// TwinCAT 3 PLC project Untitled1
// ProgramVersion: 3.1.4026.17
// libraries:
//   Tc2_Standard, * (Beckhoff Automation GmbH)
//   Tc2_System, * (Beckhoff Automation GmbH)
// project tree:
//   DUTs/ Box_Phase.TcDUT, Lay_Phase.TcDUT, Pal_Phase.TcDUT
//   GVLs/ GVL.TcGVL
//   / PlcTask.TcTTO
//   POUs/ BoxAccum.TcPOU, LayerPlace.TcPOU, MAIN.TcPOU, Pallet.TcPOU
// real-time tasks:
//   TASK PlcTask: cycle T#10ms, priority 20, ADS port 350

CONFIGURATION Untitled1
    RESOURCE PLC ON TwinCAT3
        TASK PlcTask(INTERVAL := T#10ms, PRIORITY := 20);
        PROGRAM MAIN WITH PlcTask : MAIN;
    END_RESOURCE
END_CONFIGURATION

// ---- DUTs/Box_Phase.TcDUT
{attribute 'qualified_only'}
{attribute 'strict'}
{attribute 'to_string'}
TYPE Box_Phase :
(
	Start, Run, Delay, PushFall, PushRise, TargetCheck, Clamp, Drop, Hold 
);
END_TYPE

// ---- DUTs/Lay_Phase.TcDUT
{attribute 'qualified_only'}
{attribute 'strict'}
{attribute 'to_string'}
TYPE Lay_Phase :
(
	Start,Down, LayCheck, ElvLim, ElvNex, ElvDone
):=Start;
END_TYPE

// ---- DUTs/Pal_Phase.TcDUT
{attribute 'qualified_only'}
{attribute 'strict'}
{attribute 'to_string'}
TYPE Pal_Phase :
(
	idle, Loaded, Ready_for_Boxes, Box_Loaded, Ready_for_Disp, Paused
) :=idle;
END_TYPE

// ---- GVLs/GVL.TcGVL
{attribute 'qualified_only'}
VAR_GLOBAL
    // Runtime State
    ePal_Phase              : Pal_Phase;  // Pallet machine phase
    bRunning                : BOOL;       // Line is running
    bFinishing              : BOOL;       // Graceful stop in progress
    bLayCheck               : BOOL;

    // Actuator Requests (to be AND-masked with bEnable before FIO outputs)
    // Conveyors & Belts 
    req_M010_CONV_Entry        : BOOL;
    req_M020_CONV_Incl         : BOOL;
    req_M031_CONV_PalBelt_FWD  : BOOL;
    req_M032_CONV_PalBelt_BCK  : BOOL;
    req_M080_CONV_Roll         : BOOL;
    req_M100_CONV_Exit         : BOOL;

    // Pusher / Turn / Clamp / Plate 
    req_M040_ARM_PalPush       : BOOL;
    req_M041_ARM_PalTurn       : BOOL;
    req_M050_CLAMP_Pal         : BOOL;	
    req_M050_CLAMP_Pal_B       : BOOL;
    req_M050_CLAMP_Pal_L       : BOOL;	
    req_M060_PLATE_Pal         : BOOL;     
    req_M060_PLATE_Pal_B       : BOOL;
    req_M060_PLATE_Pal_L       : BOOL;	

    // Elevator 
    req_M071_ELEV_Pal_UP       : BOOL;
    req_M072_ELEV_Pal_DOWN     : BOOL;
    req_M073_ELEV_Pal_M2LIM    : BOOL;  	
    req_M073_ELEV2TOP          : BOOL;   // move elevator to TOP 
    req_M073_ELEV2Bottom       : BOOL;   // move elevator to BOTTOM 

    // Pallet Chain
    req_M091_CONV_PalChain_FWD : BOOL;

    // Light
    req_P060_Light_SPPlus      : BOOL;   // Stack light: SP+
    req_P070_Light_SPMinus     : BOOL;   // Stack light: SP-
END_VAR

// ---- POUs/MAIN.TcPOU
PROGRAM MAIN
VAR
    // ACTUATORS (Outputs to field)
    FIO_M010_CONV_Entry          : BOOL;
    FIO_M020_CONV_Incl           : BOOL;
    FIO_M031_CONV_PalBelt_FWD    : BOOL;
    FIO_M032_CONV_PalBelt_BCK    : BOOL;
    FIO_M040_ARM_PalPush         : BOOL;
    FIO_M050_CLAMP_Pal           : BOOL;
    FIO_M060_PLATE_Pal           : BOOL;
    FIO_M071_ELEV_Pal_UP         : BOOL;
    FIO_M072_ELEV_Pal_DOWN       : BOOL;
    FIO_M073_ELEV_Pal_M2LIM      : BOOL;
    FIO_M080_CONV_Roll           : BOOL;
    FIO_M091_CONV_PalChain_FWD   : BOOL;
    FIO_M100_CONV_Exit           : BOOL;

    // SENSORS (Inputs from field)
    FIO_B010_PallClamped         : BOOL;        // Clamp sensor
    FIO_B020_PallPlateLim        : BOOL := TRUE; // NC: Plate limit (healthy=TRUE)
    FIO_B030_PallPushLim         : BOOL := TRUE; // NC: Pusher home limit (healthy=TRUE)
    FIO_B040_PallElvMov          : BOOL;        // Elevator motion status
    FIO_B050_PallElvFrLim        : BOOL;        // Elevator front/top limit
    FIO_B060_PallElvBckLim       : BOOL;        // Elevator back/bottom limit
    FIO_B070_PallReflexCnt       : BOOL := TRUE; // NC: Box counter reflex (healthy=TRUE)

    // BUTTONS 
    FIO_S100_EStop               : BOOL := TRUE; // NC: Emergency stop (healthy=TRUE)
    FIO_S010_Start               : BOOL;         // Start push button
    FIO_S020_Stop                : BOOL := TRUE; // NC: Stop push button (healthy=TRUE)
    FIO_S040_IN_LaySP_PLUS       : BOOL;         // HMI: Layer SP +
    FIO_S050_IN_LaySP_MINUS      : BOOL;         // HMI: Layer SP -

    // DISPLAYS / PROCESS VALUES (to HMI)
    // Consider RETAIN/PERSISTENT for setpoints if needed across reboots.
    FIO_P010_iPallID             : INT  := 0;   // Pallet ID
    FIO_P020_iLayCur             : INT  := 1;   // Current layer (1..10)
    FIO_P030_iLaySP              : INT  := 1;   // Layer setpoint (1..10)
    FIO_P040_Light_Start         : BOOL;        // Stack light: Start
    FIO_P050_Light_Stop          : BOOL;        // Stack light: Stop
    FIO_P060_Light_SPPlus        : BOOL;        // Stack light: SP+
    FIO_P070_Light_SPMinus       : BOOL;        // Stack light: SP-

    // FUNCTION BLOCK INSTANCES
    fbPallet		             : Pallet;
    fbBoxAccum                   : BoxAccum;
    fbLayerPlace                 : LayerPlace;


	// EDGE DETECTORS / LATCHES / FLAGS
    rStart                       : R_TRIG;      // Rising-edge detector for Start
    fStop                        : F_TRIG;      // Falling-edge detector for Stop
    fRunFall                     : F_TRIG;      // Falling-edge detector for bRunning
    srRunning                    : SR;          // Set/Reset latch for running state
    bEstopActive                 : BOOL;        // TRUE when Estop is active
END_VAR

// Structure: Safety → FBs → State → Requests → Actuators + Light

// SAFETY & RUN CONTROL
// Emergency stop
bEstopActive := NOT FIO_S100_EStop;     // TRUE = Estop pressed

// Start / Stop edge detection
rStart(CLK := FIO_S010_Start);
fStop (CLK := FIO_S020_Stop);

// SR latch for Running status
srRunning(
    SET1  := rStart.Q AND NOT bEstopActive,
    RESET := fStop.Q
);

// Running / Finishing flags 
IF srRunning.Q1 THEN
    gvl.bRunning   := TRUE;             // Enter RUN
    gvl.bFinishing := FALSE;            // Reset finishing
ELSE
    gvl.bRunning := FALSE;
END_IF

// Detect normal stop (falling edge of Running) 
fRunFall(CLK := gvl.bRunning);
IF (NOT bEstopActive) AND fRunFall.Q THEN
    gvl.bFinishing := TRUE;             // Controlled stop sequence
END_IF

//Estop clears finishing immediately
IF bEstopActive THEN
    gvl.bFinishing := FALSE;
END_IF

// FUNCTION BLOCK CALLS

fbPallet(
    PallElvFrLim := FIO_B050_PallElvFrLim,
    PallElvBckLim:= FIO_B060_PallElvBckLim,
    PallElvMov   := FIO_B040_PallElvMov,
    iPallID      => FIO_P010_iPallID
);

fbBoxAccum(
    PallClamped      := FIO_B010_PallClamped,
    PallPlateLim_NC  := FIO_B020_PallPlateLim,
    PallPushLim      := FIO_B030_PallPushLim,
    PallReflexCnt_NC := FIO_B070_PallReflexCnt
);

fbLayerPlace(
    LaySP_PLUS       := FIO_S040_IN_LaySP_PLUS,
    LaySP_MINUS      := FIO_S050_IN_LaySP_MINUS,
    PallElvMov       := FIO_B040_PallElvMov,
    iLaySP           => FIO_P030_iLaySP,
    iLayCur          => FIO_P020_iLayCur
);

// STATE → REQUESTS
// Translate pallet phase into actuator requests
CASE gvl.ePal_Phase OF

    Pal_Phase.Loaded:
        gvl.req_M073_ELEV_Pal_M2LIM := gvl.req_M073_ELEV2TOP;

    Pal_Phase.Ready_for_Boxes:
        gvl.req_M073_ELEV_Pal_M2LIM := gvl.req_M073_ELEV2Bottom;
        gvl.req_M050_CLAMP_Pal      := gvl.req_M050_CLAMP_Pal_B;
        gvl.req_M060_PLATE_Pal      := gvl.req_M050_CLAMP_Pal_B;

    Pal_Phase.Box_Loaded:
        gvl.req_M050_CLAMP_Pal      := gvl.req_M050_CLAMP_Pal_L;
        gvl.req_M060_PLATE_Pal      := gvl.req_M050_CLAMP_Pal_L;

ELSE
    gvl.req_M073_ELEV_Pal_M2LIM    := FALSE;
    gvl.req_M050_CLAMP_Pal         := FALSE;
    gvl.req_M060_PLATE_Pal         := FALSE;
END_CASE;

// REQUESTS → ACTUATORS
// Reset all outputs (avoid stale signals)
FIO_M010_CONV_Entry        := FALSE;
FIO_M020_CONV_Incl         := FALSE;
FIO_M031_CONV_PalBelt_FWD  := FALSE;
FIO_M032_CONV_PalBelt_BCK  := FALSE;
FIO_M040_ARM_PalPush       := FALSE;
FIO_M050_CLAMP_Pal         := FALSE;
FIO_M060_PLATE_Pal         := FALSE;
FIO_M071_ELEV_Pal_UP       := FALSE;
FIO_M072_ELEV_Pal_DOWN     := FALSE;
FIO_M073_ELEV_Pal_M2LIM    := FALSE;
FIO_M080_CONV_Roll         := FALSE;
FIO_M091_CONV_PalChain_FWD := FALSE;
FIO_M100_CONV_Exit         := FALSE;

// Map all requests to outputs (with Estop interlock)
FIO_M010_CONV_Entry        := gvl.req_M010_CONV_Entry        AND NOT bEstopActive;
FIO_M020_CONV_Incl         := gvl.req_M020_CONV_Incl         AND NOT bEstopActive;
FIO_M031_CONV_PalBelt_FWD  := gvl.req_M031_CONV_PalBelt_FWD  AND NOT bEstopActive;
FIO_M032_CONV_PalBelt_BCK  := gvl.req_M032_CONV_PalBelt_BCK  AND NOT bEstopActive;
FIO_M040_ARM_PalPush       := gvl.req_M040_ARM_PalPush       AND NOT bEstopActive;
FIO_M050_CLAMP_Pal         := gvl.req_M050_CLAMP_Pal         AND NOT bEstopActive;
FIO_M060_PLATE_Pal         := gvl.req_M060_PLATE_Pal         AND NOT bEstopActive;
FIO_M071_ELEV_Pal_UP       := gvl.req_M071_ELEV_Pal_UP       AND NOT bEstopActive;
FIO_M072_ELEV_Pal_DOWN     := gvl.req_M072_ELEV_Pal_DOWN     AND NOT bEstopActive;
FIO_M080_CONV_Roll         := gvl.req_M080_CONV_Roll         AND NOT bEstopActive;
FIO_M091_CONV_PalChain_FWD := gvl.req_M091_CONV_PalChain_FWD AND NOT bEstopActive;
FIO_M100_CONV_Exit         := gvl.req_M100_CONV_Exit         AND NOT bEstopActive;
FIO_M073_ELEV_Pal_M2LIM    := gvl.req_M073_ELEV_Pal_M2LIM    AND NOT bEstopActive;

// Light
FIO_P040_Light_Start       := srRunning.Q1;
FIO_P050_Light_Stop        := gvl.bFinishing;
FIO_P060_Light_SPPlus      := gvl.req_P060_Light_SPPlus;
FIO_P070_Light_SPMinus     := gvl.req_P070_Light_SPMinus;

END_PROGRAM

// ---- POUs/Pallet.TcPOU
FUNCTION_BLOCK Pallet
VAR_INPUT
    // Sensors 
    PallElvFrLim   : BOOL;   // Front limit switch
    PallElvBckLim  : BOOL;   // Back limit switch
    PallElvMov     : BOOL;   // Elevator in motion (TRUE while moving)
END_VAR

VAR_OUTPUT
    iPallID        : INT := 0;
END_VAR

VAR
    // Edge detectors
    rPallElvBckLim : R_TRIG;
    rPallElvFrLim  : R_TRIG;
    fPallElvMov    : F_TRIG;
    fPallElvFrLim  : F_TRIG;

    // Latches (SR)
    srCONV_Roll         : SR;
    srCONV_PalChain_FWD : SR;
    srELEV_Pal_UP       : SR;
END_VAR

// Edge detection 
rPallElvBckLim (CLK := PallElvBckLim);   // rising: pallet tail hits back limit
rPallElvFrLim  (CLK := PallElvFrLim);    // rising: pallet head hits front limit
fPallElvMov    (CLK := PallElvMov);      // falling: elevator motion stopped
fPallElvFrLim  (CLK := PallElvFrLim);    // falling: pallet clears front

// Safe defaults each scan
gvl.req_M080_CONV_Roll         := FALSE;
gvl.req_M091_CONV_PalChain_FWD := FALSE;    
gvl.req_M071_ELEV_Pal_UP       := FALSE;
gvl.req_M073_ELEV2TOP          := FALSE;
gvl.req_M073_ELEV_Pal_M2LIM    := FALSE;
gvl.req_M100_CONV_Exit         := FALSE;

CASE gvl.ePal_Phase OF

    // idle → load pallet
    Pal_Phase.idle:

        // Roller runs while no limits; stop on front-limit rising or stop command
        srCONV_Roll(
            SET1  := gvl.bRunning AND (NOT PallElvFrLim) AND (NOT PallElvBckLim),
            RESET := rPallElvFrLim.Q
        );
        gvl.req_M080_CONV_Roll := srCONV_Roll.Q1;
        gvl.req_M100_CONV_Exit := srCONV_Roll.Q1;

        // Chain IN: start when back-limit is hit; stop on front-limit rising or stop
        srCONV_PalChain_FWD(
            SET1  := rPallElvBckLim.Q,
            RESET := rPallElvFrLim.Q
        );
        gvl.req_M091_CONV_PalChain_FWD := srCONV_PalChain_FWD.Q1;

        // Pallet ID
        IF rPallElvBckLim.Q THEN 
            iPallID := iPallID + 10;
        END_IF

        // Transition to Loaded when both limits are TRUE
        IF PallElvFrLim AND PallElvBckLim THEN
            gvl.ePal_Phase := Pal_Phase.Loaded;
        END_IF

    // Loaded → move elevator up to the top
    Pal_Phase.Loaded:

        // Latch UP; reset when motion stops (reached top) or stop command
        srELEV_Pal_UP(
            SET1  := TRUE,       
            RESET := fPallElvMov.Q
        );
        gvl.req_M071_ELEV_Pal_UP := srELEV_Pal_UP.Q1;
        gvl.req_M073_ELEV2TOP    := srELEV_Pal_UP.Q1;   // same intent signal

        // When motion stops, elevator is at top
        IF fPallElvMov.Q THEN
            gvl.ePal_Phase := Pal_Phase.Ready_for_Boxes;
        END_IF

    // Ready_for_Boxes (no motion here)
    Pal_Phase.Ready_for_Boxes:
        // intentionally no actuator here

    // Ready_for_Disp → dispatch pallet out of the cell
    // (Phase entry is decided by the box sequence)
    Pal_Phase.Ready_for_Disp:

        // Run exit + chain only while Running
        IF gvl.bRunning THEN
            gvl.req_M100_CONV_Exit         := TRUE;
            gvl.req_M091_CONV_PalChain_FWD := TRUE;
            IF fPallElvFrLim.Q THEN
                gvl.ePal_Phase := Pal_Phase.idle;				
            END_IF
        ELSE	
            gvl.ePal_Phase := Pal_Phase.Paused;	
        END_IF

    Pal_Phase.Paused:
        IF gvl.bRunning THEN
            gvl.ePal_Phase := Pal_Phase.Ready_for_Disp;
        END_IF

ELSE
    gvl.req_M080_CONV_Roll         := FALSE;
    gvl.req_M091_CONV_PalChain_FWD := FALSE;    
    gvl.req_M071_ELEV_Pal_UP       := FALSE;
    gvl.req_M073_ELEV2TOP          := FALSE;
    gvl.req_M100_CONV_Exit         := FALSE;

END_CASE

END_FUNCTION_BLOCK

// ---- POUs/BoxAccum.TcPOU
FUNCTION_BLOCK BoxAccum
VAR_INPUT
    PallReflexCnt_NC : BOOL;   // Counting sensor: box front edge (NC type)
    PallPushLim      : BOOL;   // M040 pusher limit switch: Home=TRUE, Away=FALSE
    PallPlateLim_NC  : BOOL;   // M060 plate lower limit (NC, triggers at end of stroke)
    PallClamped      : BOOL;   // Clamp feedback signal
END_VAR

VAR_OUTPUT
END_VAR

VAR
    // Edge detection and counting 
    fBox       : F_TRIG;       // Box front edge (falling edge of NC sensor)
    CntBox     : CTU;          // Counter for boxes
    resetCnt   : BOOL;         // One-shot reset signal for counter

    // M040 pusher limits
    rPushLim   : R_TRIG;       // FALSE→TRUE : back to Home
    fPushLim   : F_TRIG;       // TRUE→FALSE : leaving Home

    // M060 plate lower limit 
    rPallPlateLim : R_TRIG;    // TRUE→FALSE (NC falling edge): plate reached open position

    // Timers
    tDelay     : TON;          // Tail-overrun delay after box arrival
    tHold      : TON;          // Hold timer for settling or confirmation

    // Phase control and target tracking
    eBP        : Box_Phase;    // Current phase/state of box accumulation process
    nextTarget : INT;          // Next counting target (e.g., 2 → 4 → 6)
END_VAR

// Defaults 
gvl.req_M010_CONV_Entry        := FALSE;
gvl.req_M020_CONV_Incl         := FALSE;
gvl.req_M031_CONV_PalBelt_FWD  := FALSE;
gvl.req_M040_ARM_PalPush       := FALSE;
gvl.req_M050_CLAMP_Pal_B       := FALSE;
gvl.req_M060_PLATE_Pal_B       := FALSE;
resetCnt                       := FALSE;

// Edge detection and counting 
fBox(CLK := PallReflexCnt_NC);

// M040 pusher (uses PallPushLim only)
rPushLim(CLK := PallPushLim);           // Back to Home (FALSE→TRUE)
fPushLim(CLK := PallPushLim);           // Leaving Home (TRUE→FALSE)

// M060 plate (uses PallPlateLim_NC only)
rPallPlateLim(CLK := PallPlateLim_NC);  // Open limit reached (NC falling edge)

// Delay timers
tDelay(IN := (eBP = Box_Phase.Delay), PT := T#1S200MS);
tHold (IN := (eBP = Box_Phase.Hold),  PT := T#200MS);  

// Phases
CASE eBP OF

    // S0: Start of a new layer
    Box_Phase.Start:
        IF gvl.bRunning 
           AND NOT gvl.req_M050_CLAMP_Pal 
           AND NOT gvl.req_M060_PLATE_Pal THEN
            nextTarget := 2;           // Target sequence: 2 → 4 → 6
            resetCnt   := TRUE;        // Reset box counter for new layer
            eBP        := Box_Phase.Run;
        END_IF;

    // S1: Feeding boxes until target count is reached
    Box_Phase.Run:
        gvl.req_M010_CONV_Entry       := TRUE;
        gvl.req_M020_CONV_Incl        := TRUE;
        gvl.req_M031_CONV_PalBelt_FWD := TRUE;

        IF CntBox.CV >= nextTarget THEN
            eBP := Box_Phase.Delay;    // Short overrun for box tail
        END_IF;

    // S2: Overrun delay (keep conveyors running briefly)
    Box_Phase.Delay:
        gvl.req_M010_CONV_Entry       := TRUE;
        gvl.req_M020_CONV_Incl        := TRUE;
        gvl.req_M031_CONV_PalBelt_FWD := TRUE;

        IF tDelay.Q THEN
            eBP := Box_Phase.PushFall; // Proceed to pusher sequence
        END_IF;

    // S3: Pusher extending – wait for “leaving Home” (TRUE→FALSE, fPushLim)
    Box_Phase.PushFall:
        gvl.req_M040_ARM_PalPush := TRUE;     
        IF fPushLim.Q THEN
            eBP := Box_Phase.PushRise; // Begin monitoring return
        END_IF;

    // S4: Pusher retracting – wait for “back to Home” (FALSE→TRUE, rPushLim)
    Box_Phase.PushRise:
        gvl.req_M040_ARM_PalPush := TRUE;     
        IF rPushLim.Q THEN
            eBP := Box_Phase.TargetCheck;
        END_IF;

    // S5: Target check
    Box_Phase.TargetCheck:
        gvl.req_M040_ARM_PalPush := FALSE;     
        IF nextTarget < 6 THEN
            nextTarget := nextTarget + 2;      // Continue with 2 → 4 → 6
            eBP        := Box_Phase.Run;
        ELSE
            eBP        := Box_Phase.Clamp;     // After 6 boxes → clamp pallet
        END_IF;

    // S6: Clamp — Clamp pallet and wait until upstream is ready
    Box_Phase.Clamp:
        gvl.req_M050_CLAMP_Pal_B := TRUE;      // Keep pallet clamped
        // Ensure pusher is at Home and conveyors stopped
        IF PallClamped 
           AND (gvl.ePal_Phase = Pal_Phase.Ready_for_Boxes) THEN
            eBP := Box_Phase.Drop;
        END_IF;

    // S7: Drop — lower plate after clamping
    Box_Phase.Drop:
        gvl.req_M050_CLAMP_Pal_B := TRUE;
        gvl.req_M060_PLATE_Pal_B := TRUE;   
        IF rPallPlateLim.Q THEN
            eBP := Box_Phase.Hold;             // Enter Hold phase 
        END_IF;

    // S8: Hold — short delay to absorb vibration
    Box_Phase.Hold:
        gvl.req_M050_CLAMP_Pal_B := TRUE;
        gvl.req_M060_PLATE_Pal_B := TRUE; 
        // Plate drive already off; maintain position for 1s
        IF tHold.Q THEN
            eBP := Box_Phase.Start;            // Return to Start for next layer
            gvl.ePal_Phase := Pal_Phase.Box_Loaded;
            gvl.bLayCheck  := TRUE;            // Mark current layer as completed
        END_IF;
END_CASE;

// Box counter (counts only when running)
CntBox(CU := fBox.Q, RESET := resetCnt, PV := 6);

END_FUNCTION_BLOCK

// ---- POUs/LayerPlace.TcPOU
FUNCTION_BLOCK LayerPlace
VAR_INPUT
    LaySP_PLUS   : BOOL;
    LaySP_MINUS  : BOOL;
    PallElvMov   : BOOL;
END_VAR

VAR_OUTPUT
    iLaySP       : INT := 1;
    iLayCur      : INT := 1;
	END_VAR
VAR
    rPlus        : R_TRIG;
    rMinus       : R_TRIG;
    rLayCheck    : R_TRIG;
    fPallElvMov  : F_TRIG;
    diff         : INT;
    eLP          : Lay_Phase;
    tHold        : TON;
END_VAR

// Edge detection 
rPlus       (CLK := LaySP_PLUS);          // Rising edge of SP+ button (increment once per press)
rMinus      (CLK := LaySP_MINUS);         // Rising edge of SP- button (decrement once per press)
fPallElvMov (CLK := PallElvMov);          // Falling edge: elevator just stopped (motion->stop)
rLayCheck   (CLK := gvl.bLayCheck);       // Rising edge: trigger for layer-check sequence

// Setpoint editing (range 1..10) 
IF rPlus.Q  AND (iLaySP < 10) THEN 
	iLaySP := iLaySP + 1; 
	gvl.req_P060_Light_SPPlus := TRUE;     // Pulse indicator for SP+
ELSE 	gvl.req_P060_Light_SPPlus := FALSE; // Otherwise keep indicator off
END_IF;

IF rMinus.Q AND (iLaySP > 1)  THEN
	iLaySP := iLaySP - 1;
	gvl.req_P070_Light_SPMinus := TRUE;    // Pulse indicator for SP- 
ELSE 	gvl.req_P070_Light_SPMinus  := FALSE;
END_IF;

// Defensive clamp for current layer (1..10)
IF iLayCur < 1 THEN
    iLayCur := 1;                          // Clamp lower bound
ELSIF iLayCur > 10 THEN
    iLayCur := 10;                         // Clamp upper bound
END_IF;

// Diff & finishing policy 
diff := iLaySP - iLayCur;                  // Positive => more layers needed
IF gvl.bFinishing THEN
    diff := 0;                             // In finishing mode, force “go to bottom” path
END_IF;

// Defaults 
gvl.req_M072_ELEV_Pal_DOWN := FALSE;       // Elevator down request (default off)
gvl.req_M073_ELEV2Bottom   := FALSE;       // “Move to bottom limit” request (default off)
gvl.req_M050_CLAMP_Pal_L   := FALSE;       // Left clamp (default off)
gvl.req_M060_PLATE_Pal_L   := FALSE;       // Left plate support (default off)

// Hold timer: active only during LayCheck to allow settling/debounce
tHold(IN := (elP = Lay_Phase.Laycheck),      PT := T#500MS);

CASE eLP OF
    Lay_Phase.Start:
        IF rLayCheck.Q THEN
            eLP := Lay_Phase.Down;             // Enter descent preparation
            gvl.bLayCheck := FALSE;            // Reset external trigger to avoid retrigger
        END_IF;

    Lay_Phase.Down:
		gvl.req_M050_CLAMP_Pal_L   := TRUE;    // Clamp pallet to reduce wobble
		gvl.req_M060_PLATE_Pal_L   := TRUE;    // Lower plate to support
        gvl.req_M072_ELEV_Pal_DOWN := TRUE;    // Request elevator down
        IF fPallElvMov.Q THEN                  // Elevator just stopped (arrived)
            eLP := Lay_Phase.Laycheck;         // Proceed to settle/check
   			gvl.ePal_Phase := Pal_Phase.Ready_for_Boxes;   // Allow box infeed on upper level
        END_IF;

    Lay_Phase.Laycheck:
	
		IF tHold.Q THEN                        // After 500 ms settle time
			  IF diff = 0 THEN
					eLP := Lay_Phase.ElvLim;     // No remaining layers → go to bottom for dispatch
				ELSE
					eLP := Lay_Phase.Start;     // Still need layers → descend one more layer
					iLayCur := iLayCur + 1;
			  END_IF;
		 END_IF;
	  
	Lay_Phase.ElvLim:
        gvl.req_M072_ELEV_Pal_DOWN := TRUE;    // Keep moving down
        gvl.req_M073_ELEV2Bottom   := TRUE;    // Command “move to bottom limit”
        IF fPallElvMov.Q THEN                  // Reached bottom (stopped)
            eLP := Lay_Phase.ElvDone;          // Ready for dispatch
        END_IF;



    Lay_Phase.ElvDone:
        gvl.ePal_Phase := Pal_Phase.Ready_for_Disp; // Elevator ready to dispatch pallet
        iLayCur := 1;                                // Reset current layer for next cycle
        eLP := Lay_Phase.Start;                      // Wait for next trigger

ELSE// Safety fallback: ensure all requests are off
    gvl.req_M072_ELEV_Pal_DOWN := FALSE;    
    gvl.req_M073_ELEV2Bottom   := FALSE;
	gvl.req_M050_CLAMP_Pal_L   := FALSE;
	gvl.req_M060_PLATE_Pal_L   := FALSE;
    eLP := Lay_Phase.Start;                 // Return to start
END_CASE;

END_FUNCTION_BLOCK
